//Provider PLC
PROGRAM MAIN
VAR
	DelayToCallInterface : UDINT := 10;
	fbDoWork			 : FB_DoWork('MAIN.fbDoWork');
END_VAR

F_ConsumeTime(DelayToCallInterface);
fbDoWork.M_Increment();

END_PROGRAM

(* stored: Version 1.1.0.1, ProductVersion 3.1.4026.18
   POU MAIN: Id {46c6155e-1631-4f07-9de1-af6d71d4f845}, SpecialFunc None *)
